// TIA Portal project "送料小车" (V17)

(* hardware
DEVICE "HMI_1"  KTP700 Basic PN
   slot 0: "HMI_1"  KTP700 Basic PN  6AV2 123-2GB03-0AX0  16.0.0.0
   slot 1: "HMI_RT_1"  KTP700 Basic PN  6AV2 123-2GB03-0AX0  16.0.0.0
   slot 5: "HMI_1.IE_CP_1"  PROFINET Interface  16.0.0.0
      slot 1: "PROFINET Interface_1"  PROFINET Interface
         slot 1: "Port_1"  Port
DEVICE "S7-1200 station_1"  S7-1200 Station
   slot 0: "Rack_0"  S7-1200 Rack  Rack  V1.0
   slot 1: "PLC_1"  CPU 1214C DC/DC/DC  6ES7 214-1AG40-0XB0  V4.5
*)

// ===== PLC "PLC_1"  CPU 1214C DC/DC/DC =====

VAR_GLOBAL   // PLC tag table "默认变量表"
   "启动按钮" AT %I0.0 : Bool;
   "停止按钮" AT %I0.1 : Bool;
   "复位按钮" AT %I0.2 : Bool;
   "原位限位开关E" AT %I0.3 : Bool;
   "卸料限位开关F" AT %I0.4 : Bool;
   "装料限位开关G" AT %I0.5 : Bool;
   "清洗限位开关H" AT %I0.6 : Bool;
   "左限限位开关K" AT %I0.7 : Bool;
   "右限限位开关L" AT %I1.0 : Bool;
   "原始位置指示灯A" AT %Q0.0 : Bool;
   "卸料处指示灯B" AT %Q0.1 : Bool;
   "装料处指示灯C" AT %Q0.2 : Bool;
   "清洗处指示灯D" AT %Q0.3 : Bool;
   "正转" AT %Q0.4 : Bool;
   "反转" AT %Q0.5 : Bool;
   "启动线圈" AT %M0.0 : Bool;
   "停止线圈" AT %M0.1 : Bool;
   "启动按钮触摸屏" AT %M0.2 : Bool;
   "停止按钮触摸屏" AT %M0.3 : Bool;
   "复位按钮触摸屏" AT %M0.4 : Bool;
   "“原位装料”控制" AT %M0.5 : Bool;
   "原始限位开关E触摸屏" AT %M0.6 : Bool;
   "卸料限位开关F触摸屏" AT %M0.7 : Bool;
   "装料限位开关G触摸屏" AT %M1.0 : Bool;
   "清洗限位开关H触摸屏" AT %M1.1 : Bool;
   "卸料限位开关F线圈" AT %M1.2 : Bool;
   "装料限位开关G线圈" AT %M1.3 : Bool;
   "清洗限位开关H线圈" AT %M1.4 : Bool;
   "原料装料" AT %M1.5 : Bool;
   "装料卸料" AT %M1.6 : Bool;
   "卸料清洗" AT %M1.7 : Bool;
   "清洗装料" AT %M2.0 : Bool;
   "清洗原位" AT %M2.1 : Bool;
   "上升沿检测存储" AT %M2.2 : Bool;
   "时钟存储1" AT %M2.3 : Bool;
   "时钟存储2" AT %M2.4 : Bool;
   "小车移动距离" AT %MW100 : Word;
   "Clock_Byte" AT %MB13 : Byte;
   "Clock_10Hz" AT %M13.0 : Bool;
   "Clock_5Hz" AT %M13.1 : Bool;
   "Clock_2.5Hz" AT %M13.2 : Bool;
   "Clock_2Hz" AT %M13.3 : Bool;
   "Clock_1.25Hz" AT %M13.4 : Bool;
   "Clock_1Hz" AT %M13.5 : Bool;
   "Clock_0.625Hz" AT %M13.6 : Bool;
   "Clock_0.5Hz" AT %M13.7 : Bool;
END_VAR

// folder: System blocks/Program resources

DATA_BLOCK "T1"   // DB1
{ S7_Optimized_Access := 'TRUE' }
AUTHOR : Simatic
FAMILY : IEC
NAME : IEC_TMR
VERSION : 1.0
// stored: InstanceOfName IEC_TIMER
"IEC_TIMER"
BEGIN
END_DATA_BLOCK

DATA_BLOCK "T2"   // DB2
{ S7_Optimized_Access := 'TRUE' }
AUTHOR : Simatic
FAMILY : IEC
NAME : IEC_TMR
VERSION : 1.0
// stored: InstanceOfName IEC_TIMER
"IEC_TIMER"
BEGIN
END_DATA_BLOCK

DATA_BLOCK "T3"   // DB3
{ S7_Optimized_Access := 'TRUE' }
AUTHOR : Simatic
FAMILY : IEC
NAME : IEC_TMR
VERSION : 1.0
// stored: InstanceOfName IEC_TIMER
"IEC_TIMER"
BEGIN
END_DATA_BLOCK

// folder: (top level)

ORGANIZATION_BLOCK "Main"   // OB1, LAD, ProgramCycle
TITLE = "Main Program Sweep (Cycle)"
{ S7_Optimized_Access := 'TRUE' }
VERSION : 0.1
   VAR_INPUT
      Initial_Call : Bool;   // Initial call of this OB
      Remanence : Bool;   // =True, if remanent data are available
   END_VAR
   VAR_TEMP   // added for the SCL form of the ladder/FBD networks
      _w1 : Bool;
   END_VAR
BEGIN

REGION Network 1
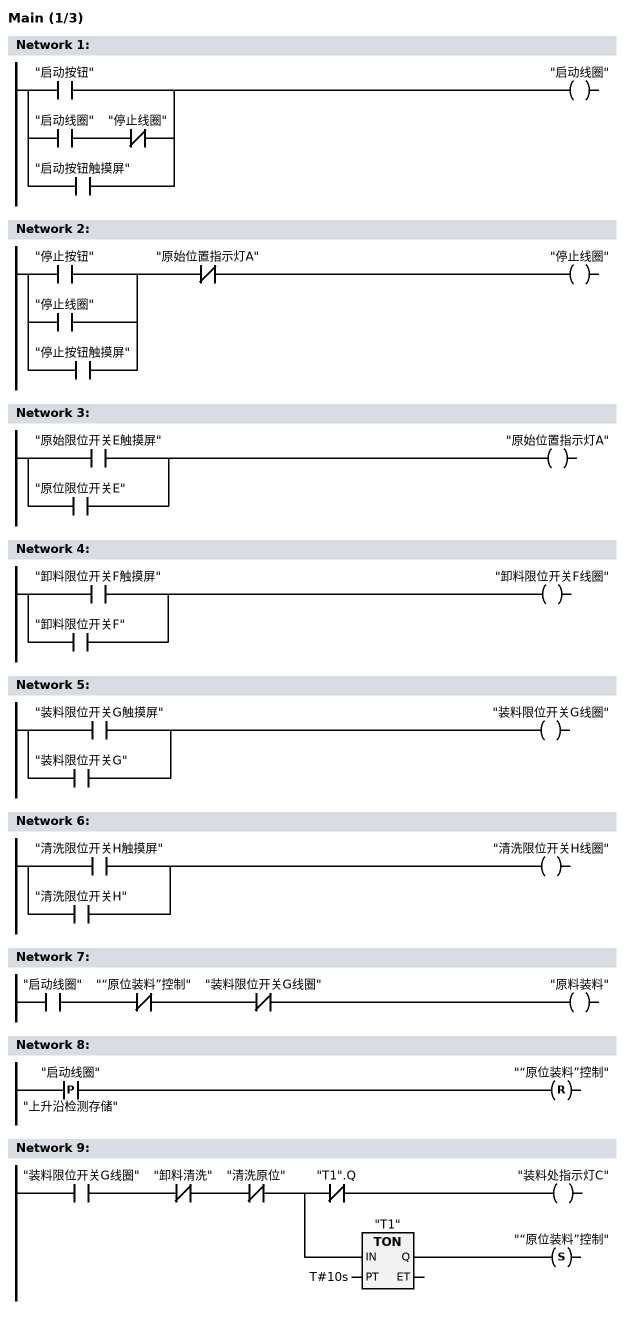
   RUNG wire#powerrail
      Contact( "启动按钮" )
      wire#w1
      Coil( "启动线圈" )
   END_RUNG
   RUNG wire#powerrail
      Contact( "启动线圈" )
      I_Contact( "停止线圈" )
   END_RUNG wire#w1
   RUNG wire#powerrail
      Contact( "启动按钮触摸屏" )
   END_RUNG wire#w1
   // the same network as SCL:
   "启动线圈" := "启动按钮" OR ("启动线圈" AND NOT "停止线圈") OR "启动按钮触摸屏";
END_REGION

REGION Network 2
   RUNG wire#powerrail
      Contact( "停止按钮" )
      wire#w1
      I_Contact( "原始位置指示灯A" )
      Coil( "停止线圈" )
   END_RUNG
   RUNG wire#powerrail
      Contact( "停止线圈" )
   END_RUNG wire#w1
   RUNG wire#powerrail
      Contact( "停止按钮触摸屏" )
   END_RUNG wire#w1
   // the same network as SCL:
   "停止线圈" := ("停止按钮" OR "停止线圈" OR "停止按钮触摸屏") AND NOT "原始位置指示灯A";
END_REGION

REGION Network 3
   RUNG wire#powerrail
      Contact( "原始限位开关E触摸屏" )
      wire#w1
      Coil( "原始位置指示灯A" )
   END_RUNG
   RUNG wire#powerrail
      Contact( "原位限位开关E" )
   END_RUNG wire#w1
   // the same network as SCL:
   "原始位置指示灯A" := "原始限位开关E触摸屏" OR "原位限位开关E";
END_REGION

REGION Network 4
   RUNG wire#powerrail
      Contact( "卸料限位开关F触摸屏" )
      wire#w1
      Coil( "卸料限位开关F线圈" )
   END_RUNG
   RUNG wire#powerrail
      Contact( "卸料限位开关F" )
   END_RUNG wire#w1
   // the same network as SCL:
   "卸料限位开关F线圈" := "卸料限位开关F触摸屏" OR "卸料限位开关F";
END_REGION

REGION Network 5
   RUNG wire#powerrail
      Contact( "装料限位开关G触摸屏" )
      wire#w1
      Coil( "装料限位开关G线圈" )
   END_RUNG
   RUNG wire#powerrail
      Contact( "装料限位开关G" )
   END_RUNG wire#w1
   // the same network as SCL:
   "装料限位开关G线圈" := "装料限位开关G触摸屏" OR "装料限位开关G";
END_REGION

REGION Network 6
   RUNG wire#powerrail
      Contact( "清洗限位开关H触摸屏" )
      wire#w1
      Coil( "清洗限位开关H线圈" )
   END_RUNG
   RUNG wire#powerrail
      Contact( "清洗限位开关H" )
   END_RUNG wire#w1
   // the same network as SCL:
   "清洗限位开关H线圈" := "清洗限位开关H触摸屏" OR "清洗限位开关H";
END_REGION

REGION Network 7
   RUNG wire#powerrail
      Contact( "启动线圈" )
      I_Contact( "“原位装料”控制" )
      I_Contact( "装料限位开关G线圈" )
      Coil( "原料装料" )
   END_RUNG
   // the same network as SCL:
   "原料装料" := "启动线圈" AND NOT "“原位装料”控制" AND NOT "装料限位开关G线圈";
END_REGION

REGION Network 8
   RUNG wire#powerrail
      P_Contact(operand := "启动线圈", bit := "上升沿检测存储")
      R_Coil( "“原位装料”控制" )
   END_RUNG
   // the same network as SCL:
   #_w1 := "启动线圈" AND NOT "上升沿检测存储";   // rising edge of "启动线圈"
   "上升沿检测存储" := "启动线圈";
   IF #_w1 THEN "“原位装料”控制" := FALSE; END_IF;
END_REGION

REGION Network 9
   #_w1 := "装料限位开关G线圈" AND NOT "卸料清洗" AND NOT "清洗原位";
   "装料处指示灯C" := #_w1 AND NOT "T1".Q;
   "T1".TON(IN := #_w1, PT := T#10s);
   IF "T1".Q THEN "“原位装料”控制" := TRUE; END_IF;
END_REGION

REGION Network 10
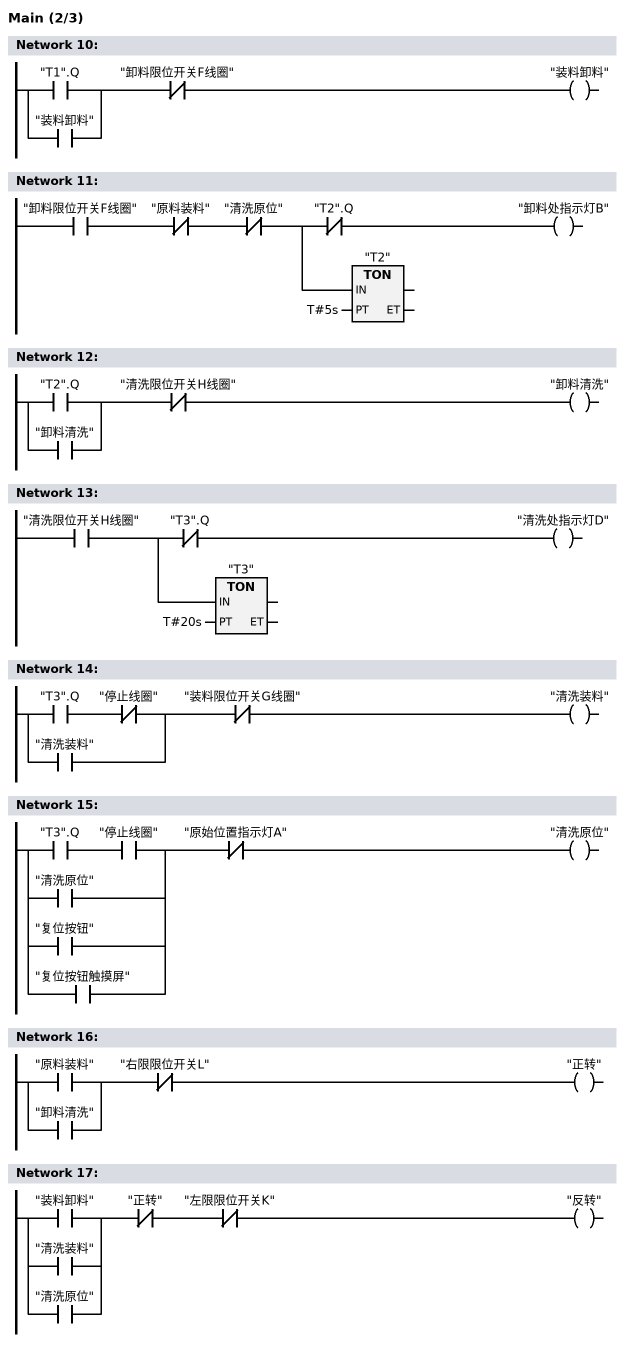
   RUNG wire#powerrail
      Contact( "T1".Q )
      wire#w1
      I_Contact( "卸料限位开关F线圈" )
      Coil( "装料卸料" )
   END_RUNG
   RUNG wire#powerrail
      Contact( "装料卸料" )
   END_RUNG wire#w1
   // the same network as SCL:
   "装料卸料" := ("T1".Q OR "装料卸料") AND NOT "卸料限位开关F线圈";
END_REGION

REGION Network 11
   #_w1 := "卸料限位开关F线圈" AND NOT "原料装料" AND NOT "清洗原位";
   "卸料处指示灯B" := #_w1 AND NOT "T2".Q;
   "T2".TON(IN := #_w1, PT := T#5s);
END_REGION

REGION Network 12
   RUNG wire#powerrail
      Contact( "T2".Q )
      wire#w1
      I_Contact( "清洗限位开关H线圈" )
      Coil( "卸料清洗" )
   END_RUNG
   RUNG wire#powerrail
      Contact( "卸料清洗" )
   END_RUNG wire#w1
   // the same network as SCL:
   "卸料清洗" := ("T2".Q OR "卸料清洗") AND NOT "清洗限位开关H线圈";
END_REGION

REGION Network 13
   "清洗处指示灯D" := "清洗限位开关H线圈" AND NOT "T3".Q;
   "T3".TON(IN := "清洗限位开关H线圈", PT := T#20s);
END_REGION

REGION Network 14
   RUNG wire#powerrail
      Contact( "T3".Q )
      I_Contact( "停止线圈" )
      wire#w1
      I_Contact( "装料限位开关G线圈" )
      Coil( "清洗装料" )
   END_RUNG
   RUNG wire#powerrail
      Contact( "清洗装料" )
   END_RUNG wire#w1
   // the same network as SCL:
   "清洗装料" := (("T3".Q AND NOT "停止线圈") OR "清洗装料") AND NOT "装料限位开关G线圈";
END_REGION

REGION Network 15
   RUNG wire#powerrail
      Contact( "T3".Q )
      Contact( "停止线圈" )
      wire#w1
      I_Contact( "原始位置指示灯A" )
      Coil( "清洗原位" )
   END_RUNG
   RUNG wire#powerrail
      Contact( "清洗原位" )
   END_RUNG wire#w1
   RUNG wire#powerrail
      Contact( "复位按钮" )
   END_RUNG wire#w1
   RUNG wire#powerrail
      Contact( "复位按钮触摸屏" )
   END_RUNG wire#w1
   // the same network as SCL:
   "清洗原位" := (("T3".Q AND "停止线圈") OR "清洗原位" OR "复位按钮" OR "复位按钮触摸屏") AND NOT "原始位置指示灯A";
END_REGION

REGION Network 16
   RUNG wire#powerrail
      Contact( "原料装料" )
      wire#w1
      I_Contact( "右限限位开关L" )
      Coil( "正转" )
   END_RUNG
   RUNG wire#powerrail
      Contact( "卸料清洗" )
   END_RUNG wire#w1
   // the same network as SCL:
   "正转" := ("原料装料" OR "卸料清洗") AND NOT "右限限位开关L";
END_REGION

REGION Network 17
   RUNG wire#powerrail
      Contact( "装料卸料" )
      wire#w1
      I_Contact( "正转" )
      I_Contact( "左限限位开关K" )
      Coil( "反转" )
   END_RUNG
   RUNG wire#powerrail
      Contact( "清洗装料" )
   END_RUNG wire#w1
   RUNG wire#powerrail
      Contact( "清洗原位" )
   END_RUNG wire#w1
   // the same network as SCL:
   "反转" := ("装料卸料" OR "清洗装料" OR "清洗原位") AND NOT "正转" AND NOT "左限限位开关K";
END_REGION

REGION Network 18
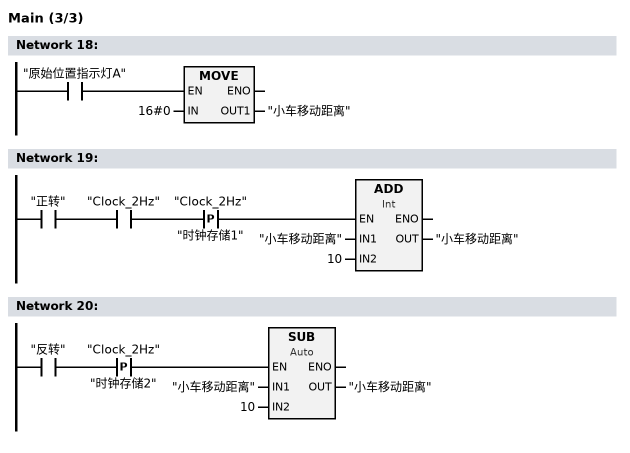
   RUNG wire#powerrail
      Contact( "原始位置指示灯A" )
      Move(in := 16#0, out1 => "小车移动距离")
   END_RUNG
   // the same network as SCL:
   IF "原始位置指示灯A" THEN "小车移动距离" := 16#0; END_IF;
END_REGION

REGION Network 19
   RUNG wire#powerrail
      Contact( "正转" )
      Contact( "Clock_2Hz" )
      P_Contact(operand := "Clock_2Hz", bit := "时钟存储1")
      { S7_Templates := "SrcType := Int" } Add(in1 := "小车移动距离", in2 := 10, out => "小车移动距离")
   END_RUNG
   // the same network as SCL:
   #_w1 := "正转" AND "Clock_2Hz" AND "Clock_2Hz" AND NOT "时钟存储1";   // rising edge of "Clock_2Hz"
   "时钟存储1" := "Clock_2Hz";
   IF #_w1 THEN "小车移动距离" := "小车移动距离" + 10; END_IF;
END_REGION

REGION Network 20
   RUNG wire#powerrail
      Contact( "反转" )
      P_Contact(operand := "Clock_2Hz", bit := "时钟存储2")
      Sub(in1 := "小车移动距离", in2 := 10, out => "小车移动距离")
   END_RUNG
   // the same network as SCL:
   #_w1 := "反转" AND "Clock_2Hz" AND NOT "时钟存储2";   // rising edge of "Clock_2Hz"
   "时钟存储2" := "Clock_2Hz";
   IF #_w1 THEN "小车移动距离" := "小车移动距离" - 10; END_IF;
END_REGION
END_ORGANIZATION_BLOCK

(* ===== HMI "HMI_RT_1" =====
system functions are stored by id; their names below are inferred from use
connection "HMI_连接_1": ETHERNET, SMART_S7_1200_OMS

HMI tags "默认变量表"
   "启动按钮触摸屏" : Bool = PLC 启动按钮触摸屏 AT %M0.2, 1 s
   "停止按钮触摸屏" : Bool = PLC 停止按钮触摸屏 AT %M0.3, 1 s
   "复位按钮触摸屏" : Bool = PLC 复位按钮触摸屏 AT %M0.4, 1 s
   "装料限位开关G触摸屏" : Bool = PLC 装料限位开关G触摸屏 AT %M1.0, 1 s
   "卸料限位开关F触摸屏" : Bool = PLC 卸料限位开关F触摸屏 AT %M0.7, 1 s
   "原始限位开关E触摸屏" : Bool = PLC 原始限位开关E触摸屏 AT %M0.6, 1 s
   "反转" : Bool = PLC 反转 AT %Q0.5, 1 s
   "正转" : Bool = PLC 正转 AT %Q0.4, 1 s
   "原位限位指示灯A" : Bool = PLC 原始位置指示灯A AT %Q0.0, 1 s
   "卸料处指示灯B" : Bool = PLC 卸料处指示灯B AT %Q0.1, 1 s
   "装料处指示灯C" : Bool = PLC 装料处指示灯C AT %Q0.2, 1 s
   "清洗处指示灯D" : Bool = PLC 清洗处指示灯D AT %Q0.3, 1 s
   "小车移动距离" : Word = PLC 小车移动距离 AT %MW100, 1 s
   "清洗限位开关H触摸屏" : Bool = PLC 清洗限位开关H触摸屏 AT %M1.1, 1 s

screen "画面_1" 800x480
   Circle "圆_1" at 49,69 size 48x48
      Appearance <- "正转"
   Circle "圆_3" at 49,136 size 48x48
      Appearance <- "反转"
   Circle "圆_4" at 505,344 size 48x48
      Appearance <- "清洗处指示灯D"
   Circle "圆_5" at 398,344 size 48x48
      Appearance <- "装料处指示灯C"
   Circle "圆_6" at 289,344 size 48x48
      Appearance <- "卸料处指示灯B"
   Circle "圆_7" at 182,344 size 48x48
      Appearance <- "原位限位指示灯A"
   Button "按钮_1" at 537,69 size 96x32; TextOff '启动'
      on Release: ResetBit("启动按钮触摸屏")
      on Press: SetBit("启动按钮触摸屏")
   Button "按钮_2" at 537,124 size 96x32; TextOff '停止'
      on Release: ResetBit("停止按钮触摸屏")
      on Press: SetBit("停止按钮触摸屏")
   Button "按钮_3" at 537,171 size 96x32; TextOff '复位'
      on Release: ResetBit("复位按钮触摸屏")
      on Press: SetBit("复位按钮触摸屏")
   Button "按钮_4" at 156,404 size 96x32; TextOff '原位'
      on Release: ResetBit("原始限位开关E触摸屏")
      on Press: SetBit("原始限位开关E触摸屏")
   Button "按钮_5" at 266,405 size 96x32; TextOff '卸料'
      on Release: ResetBit("卸料限位开关F触摸屏")
      on Press: SetBit("卸料限位开关F触摸屏")
   Button "按钮_6" at 375,405 size 96x32; TextOff '装料'
      on Release: ResetBit("装料限位开关G触摸屏")
      on Press: SetBit("装料限位开关G触摸屏")
   Button "按钮_7" at 482,405 size 96x32; TextOff '清洗'
      on Release: ResetBit("清洗限位开关H触摸屏")
      on Press: SetBit("清洗限位开关H触摸屏")
   Group "Group" at 181,275 size 55x52
      HorizontalMovement <- "小车移动距离"
   TextField "文本域_1" at 127,77 size 53x27; Text '正转'
   TextField "文本域_2" at 128,149 size 53x27; Text '反转'
   TextField "文本域_3" at 251,18 size 201x52; Text '送料小车'
*)